FUNCTION_BLOCK FB_CAMERA_DiagnosticLog
VAR_INPUT
	bLogData			: BOOL;
	nExpectedResp		: INT;
	bAddScanNo			: BOOL;
END_VAR
VAR_IN_OUT
	stCameraStatus		: ST_CAMERA_Status;
END_VAR
VAR_OUTPUT
	sCodeDiagnostig		: T_LongSTRING;
END_VAR
VAR
	rtExecute			: R_TRIG;
	nIndex				: INT;
	sAppendedString		: STRING;
END_VAR

rtExecute(CLK:=bLogData);

IF rtExecute.Q THEN
	
	sAppendedString	:= '';
	sCodeDiagnostig	:= '';
	
	IF bAddScanNo THEN
		CONCAT2(ADR(sCodeDiagnostig), ADR('['), ADR(sCodeDiagnostig), SIZEOF(sCodeDiagnostig));
		sAppendedString := INT_TO_STRING(stCameraStatus.I.stTriggerID.nScanNo);
		CONCAT2(ADR(sCodeDiagnostig), ADR(sAppendedString), ADR(sCodeDiagnostig), SIZEOF(sCodeDiagnostig));
		CONCAT2(ADR(sCodeDiagnostig), ADR('] - '), ADR(sCodeDiagnostig), SIZEOF(sCodeDiagnostig));
	END_IF
	
	CONCAT2(ADR(sCodeDiagnostig), ADR(stCameraStatus.Q.stImageData.aCodeData[1].sDataString), ADR(sCodeDiagnostig), SIZEOF(sCodeDiagnostig));
	CONCAT2(ADR(sCodeDiagnostig), ADR(' [PN:'), ADR(sCodeDiagnostig), SIZEOF(sCodeDiagnostig));
	sAppendedString := BYTE_TO_STRING(stCameraStatus.Q.stImageData.aCodeData[1].nProgramNo);
	CONCAT2(ADR(sCodeDiagnostig), ADR(sAppendedString), ADR(sCodeDiagnostig), SIZEOF(sCodeDiagnostig));
	CONCAT2(ADR(sCodeDiagnostig), ADR(']'), ADR(sCodeDiagnostig), SIZEOF(sCodeDiagnostig));
	
	IF nExpectedResp > 1 THEN
		FOR nIndex := 2 TO nExpectedResp BY 1 DO
				
			CONCAT2(ADR(sCodeDiagnostig), ADR(' - '), ADR(sCodeDiagnostig), SIZEOF(sCodeDiagnostig));
			CONCAT2(ADR(sCodeDiagnostig), ADR(stCameraStatus.Q.stImageData.aCodeData[nIndex].sDataString), ADR(sCodeDiagnostig), SIZEOF(sCodeDiagnostig));
			CONCAT2(ADR(sCodeDiagnostig), ADR(' [PN:'), ADR(sCodeDiagnostig), SIZEOF(sCodeDiagnostig));
			sAppendedString := BYTE_TO_STRING(stCameraStatus.Q.stImageData.aCodeData[nIndex].nProgramNo);
			CONCAT2(ADR(sCodeDiagnostig), ADR(sAppendedString), ADR(sCodeDiagnostig), SIZEOF(sCodeDiagnostig));
			CONCAT2(ADR(sCodeDiagnostig), ADR(']'), ADR(sCodeDiagnostig), SIZEOF(sCodeDiagnostig));
	
		END_FOR
	END_IF
END_IF

END_FUNCTION_BLOCK

(* stored: Version 1.1.0.1
   POU FB_CAMERA_DiagnosticLog: Id {b0ea89d9-8c18-479b-93ac-fb3f3183b348}, SpecialFunc None *)
